# EPICS autosave request: aliveApp/Db/aliveMSGCalc_local.req
file calcout_settings.req P=$(P)aliveMSGCalc
